// TIA Portal V16 export
// export: Created 2023-07-30T20:35:43.0210697Z, ExportSetting WithDefaults, DisplayName Totally Integrated Automation Portal, DisplayVersion V16, DisplayName TIA Portal Version Control Interface, DisplayVersion V16, DisplayName TIA Portal Openness, DisplayVersion V16, DisplayName STEP 7 Professional, DisplayVersion V16, DisplayName STEP 7 Safety, DisplayVersion V16, DisplayName WinCC Professional, DisplayVersion V16
VAR_GLOBAL   // PLC tag table "Default tag table"
   System_Byte AT %MB100 : Byte;
   FirstScan AT %M100.0 : Bool;
   DiagStatusUpdate AT %M100.1 : Bool;
   AlwaysTRUE AT %M100.2 : Bool;
   AlwaysFALSE AT %M100.3 : Bool;
   "System_Byte(1)" AT %MB1 : Byte;
   Clock_Byte AT %MB101 : Byte;
   Clock_10Hz AT %M101.0 : Bool;
   Clock_5Hz AT %M101.1 : Bool;
   "Clock_2.5Hz" AT %M101.2 : Bool;
   Clock_2Hz AT %M101.3 : Bool;
   "Clock_1.25Hz" AT %M101.4 : Bool;
   Clock_1Hz AT %M101.5 : Bool;
   "Clock_0.625Hz" AT %M101.6 : Bool;
   "Clock_0.5Hz" AT %M101.7 : Bool;
END_VAR
